// TIA Portal V17 export
// export: Created 2023-02-13T11:16:41.5834687Z, ExportSetting WithDefaults, DisplayName Totally Integrated Automation Portal, DisplayVersion V17, DisplayName TIA Portal Openness, DisplayVersion V17, DisplayName TIA Portal Teamcenter Gateway, DisplayVersion V17, DisplayName TIA Portal Version Control Interface, DisplayVersion V17, DisplayName SINAMICS Startdrive Advanced, DisplayVersion V17, DisplayName SINAMICS Startdrive G130, G150, S120, S150, SINAMICS MV, S210, DisplayVersion V17, DisplayName SINAMICS Startdrive G110M, G120, G120C, G120D, G120P, G115D, DisplayVersion V17, DisplayName STEP 7 Professional, DisplayVersion V17, DisplayName STEP 7 Safety, DisplayVersion V17, DisplayName WinCC Professional, DisplayVersion V17
DATA_BLOCK "General Preparation"   // DB59
{ S7_Optimized_Access := 'TRUE' }
VERSION : 0.1
// stored: AutoNumber true, DBAccessibleFromOPCUA true, DBAccessibleFromWebserver true, IsOnlyStoredInLoadMemory false, IsRetainMemResEnabled false, IsWriteProtectedInAS false, MemoryReserve 100
   VAR
      "Header 1" : Struct
         "CIP Enable" : Bool;
         "CIP Request" : Bool;
         "CIP Line OK" : Bool;
         "CIP on Prog" : Bool;
         V_CIP_Cmd : Bool;
         p_trig : Bool;
      END_STRUCT;
      "Header 2" : Struct
         "CIP Enable" : Bool;
         "CIP Request" : Bool;
         "CIP Line OK" : Bool;
         "CIP on Prog" : Bool;
         V_CIP_Cmd : Bool;
         p_trig : Bool;
      END_STRUCT;
      "Blend OSA" : Struct
         "CIP Enable_T-06 Cmd" : Bool;
         "CIP Enable_T-07 Cmd" : Bool;
         "CIP Enable_T-08 Cmd" : Bool;
         "CIP Request" : Bool;
         "CIP on Prog" : Bool;
         "CIP EN T-06" : Bool;
         "CIP EN T-07" : Bool;
         "CIP EN T-08" : Bool;
      END_STRUCT;
      "Tipper 1" : Struct
         "CIP Enable Cmd" : Bool;
         "CIP Request" : Bool;
         "CIP on Prog" : Bool;
         "CIP EN" : Bool;
      END_STRUCT;
      "Tipper 2" : Struct
         "CIP Enable_T-03 Cmd" : Bool;
         "CIP Enable_T-04 Cmd" : Bool;
         "CIP Request" : Bool;
         "CIP on Prog" : Bool;
         "CIP EN T-03" : Bool;
         "CIP EN T-04" : Bool;
      END_STRUCT;
      CIP_Bypass : Bool;
      Reset_Totalizer : Struct
         "FT_T-51" : Bool;
         "FT_T-02" : Bool;
         "FT_T-3" : Bool;
         "FT_T-4" : Bool;
         "FT_T-5" : Bool;
         "FT_T-6" : Bool;
         "FT_T-7" : Bool;
         "FT_T-8" : Bool;
         "FT_T-9" : Bool;
         "FT_T-10" : Bool;
      END_STRUCT;
      CV_Value_Manual : Real;
   END_VAR
   VAR RETAIN
      Tank_Name : Struct
         ChiliAwetan1 : String := 'Chili Awetan 1';
         ChiliAwetan2 : String := 'Chili Awetan 2';
         ChiliAwetan3 : String := 'Chili Awetan 3';
         Tomato : String := 'Tomato';
         ChiliFresh1 : String := 'Chili Fresh 1';
         ChiliFresh2 : String := 'Chili Fresh 2';
         ChiliFresh3 : String := 'Chili Fresh 3';
         Garlic : String := 'Garlic';
         Vinegar : String := 'Vinegar';
         HotWater : String := 'Hot Water';
         free11 : String;
      END_STRUCT;
   END_VAR
BEGIN
END_DATA_BLOCK
